{attribute 'qualified_only'}
{attribute 'strict'}
TYPE E_AxisDirection :
(
	eForward := 0,
	eBackward := 1
);
END_TYPE

(* stored: Version 1.1.0.1
   DUT E_AxisDirection: Id {aa0c8317-f76e-0c52-03ff-32ef6f937332} *)
